{attribute 'linkalways'} 
{attribute 'no_explicit_call' := 'This FB is a CLASS and must be accessed using methods or properties'}
{attribute 'enable_dynamic_creation'}
FUNCTION_BLOCK PUBLIC DefaultPositionHomeBuilder IMPLEMENTS PositionHomeBuilder
VAR
	parent_builder : POINTER TO DefaultHomeBuilder;
END_VAR

METHOD PUBLIC BufferMode : PositionHomeBuilder
VAR_INPUT
	value : MotionBufferMode;
END_VAR
parent_builder^.BufferMode(value);
BufferMode := THIS^;
END_METHOD

METHOD PUBLIC BuildDefaultHomingCommand : AsyncCommand
VAR_INPUT
	axis : Axis;
END_VAR
BuildDefaultHomingCommand := parent_builder^.BuildDefaultHomingCommand(axis);
END_METHOD

METHOD PUBLIC BuildDirectCommand : AsyncCommand
VAR_INPUT
	axis : Axis;
END_VAR
BuildDirectCommand := parent_builder^.BuildDirectCommand(axis);
END_METHOD

//FB_Init is always available implicitly and it is used primarily for initialization.
//The return value is not evaluated. For a specific influence, you can also declare the
//methods explicitly and provide additional code there with the standard initialization
//code. You can evaluate the return value.
METHOD FB_Init: BOOL
VAR_INPUT
    bInitRetains : BOOL; // TRUE: the retain variables are initialized (reset warm / reset cold)
    bInCopyCode : BOOL;  // TRUE: the instance will be copied to the copy code afterward (online change)
	parent_builder : POINTER TO DefaultHomeBuilder;
END_VAR
THIS^.parent_builder := parent_builder;
END_METHOD

METHOD PUBLIC Position : PositionHomeBuilder
VAR_INPUT
	value : LREAL;
END_VAR
parent_builder^.Position(value);
Position := THIS^;
END_METHOD

METHOD PUBLIC Reset : PositionHomeBuilder
parent_builder^.Reset();
Reset := THIS^;
END_METHOD

METHOD PUBLIC SearchDirection : PositionHomeBuilder
VAR_INPUT
	value : MotionDirection;
END_VAR
parent_builder^.SearchDirection(value);
SearchDirection := THIS^;
END_METHOD

METHOD PUBLIC SearchVelocity : PositionHomeBuilder
VAR_INPUT
	value : LREAL;
END_VAR
parent_builder^.SearchVelocity(value);
SearchVelocity := THIS^;
END_METHOD

METHOD PUBLIC SyncDirection : PositionHomeBuilder
VAR_INPUT
	value : MotionDirection;
END_VAR
parent_builder^.SyncDirection(value);
SyncDirection := THIS^;
END_METHOD

METHOD PUBLIC SyncVelocity : PositionHomeBuilder
VAR_INPUT
	value : LREAL;
END_VAR
parent_builder^.SyncVelocity(value);
SyncVelocity := THIS^;
END_METHOD

END_FUNCTION_BLOCK

(* stored: Version 1.1.0.1
   POU DefaultPositionHomeBuilder: Id {9ac5065d-39be-47dc-b401-3d34da0b4668}, SpecialFunc None
   Folder Builders: Id {a726cef4-397b-40cf-a475-dda7f232e823}
   Folder Constructor: Id {b0a213a6-7fae-4d5a-99b7-4017c216fa89}
   Folder PropertySetters: Id {26713346-d1d5-4f9c-be63-0d58882afba2}
   Method BufferMode: Id {792c58fb-f6aa-4c00-a2b3-b735a5da0c84}
   Method BuildDefaultHomingCommand: Id {318cb9b1-afef-432f-955e-92bece71935c}
   Method BuildDirectCommand: Id {c30b933c-957e-4ad3-b157-5f975a195d4d}
   Method FB_Init: Id {c84ce3ed-954d-45be-9b9d-454884e16913}
   Method Position: Id {f41ff002-e811-444c-8c53-0888f801889f}
   Method Reset: Id {166b9989-7dbc-4bce-a082-ec32d1f63d2d}
   Method SearchDirection: Id {46d1416a-d5a0-4f06-ad89-8dfa1125369e}
   Method SearchVelocity: Id {c13553c3-666b-4c94-ad18-04e377ddb547}
   Method SyncDirection: Id {9486fbfe-b113-411b-9aa3-1434b9e10d31}
   Method SyncVelocity: Id {eaeed09e-c57a-46a9-b5f1-61bdcb0b6061} *)
